// TwinCAT 3 PLC project database_connection
// Title: cyclic_database_recorder
// Company: Beckhoff K.K. - Japan
// Author: Takashi Ichihashi
// ProjectVersion: 1.0.1.1
// Description: The database recording library for InfluxDB. Requirements: Tc2_Utilities / T_Arg function
// ProgramVersion: 3.1.4023.0
// libraries:
//   Tc2_EtherCAT, * (Beckhoff Automation GmbH)
//   Tc2_Standard, * (Beckhoff Automation GmbH)
//   Tc2_System, * (Beckhoff Automation GmbH)
//   Tc2_Utilities, * (Beckhoff Automation GmbH)
//   Tc3_Database, * (Beckhoff Automation GmbH)
//   Tc3_IPCDiag, * (Beckhoff Automation GmbH)
//   Tc3_Module, * (Beckhoff Automation GmbH)
// project tree:
//   / DBWrite.TcTTO, PlcTask.TcTTO
//   DUTs/ ChunkCommand.TcDUT, DatabaseThroughput.TcDUT, DatabaseThroughput_SQL.TcDUT, DataTag.TcDUT, E_DbLogState.TcDUT, PerformanceData.TcDUT, ProcessModeData.TcDUT, RecordDataStructureInfo.TcDUT, SQLPerformanceData.TcDUT
//   GVLs/ GVL.TcGVL, DBLibParam.TcGVL
//   POUs/ DatabaseRecord.TcPOU, SampleProgram.TcPOU
//   POUs/library/ BufferedRecord.TcPOU, dequeue.TcPOU
//   POUs/library/InfluxDB/ InfluxdbMeasurement.TcPOU, RecordInfluxDB.TcPOU
//   POUs/library/interface/ IRecordDataQueue.TcIO, IRecordDB.TcIO
//   POUs/library/SQL/ FB_DatetimeUtilities.TcPOU, sql_parameters.TcPOU, RecordSQL.TcPOU
//   Project Information/ F_GetCompany.TcPOU, F_GetTitle.TcPOU, F_GetVersion.TcPOU
//   Version/ Global_Version.TcGVL
// real-time tasks:
//   TASK PlcTask: cycle T#1ms, priority 20, ADS port 350
//   TASK DBWrite: cycle T#10ms, priority 1, ADS port 351

CONFIGURATION database_connection
    RESOURCE PLC ON TwinCAT3
        TASK DBWrite(INTERVAL := T#10ms, PRIORITY := 1);
        TASK PlcTask(INTERVAL := T#1ms, PRIORITY := 20);
        PROGRAM DatabaseRecord WITH DBWrite : DatabaseRecord;
        PROGRAM SampleProgram WITH PlcTask : SampleProgram;
    END_RESOURCE
END_CONFIGURATION

// ---- DUTs/ChunkCommand.TcDUT
TYPE ChunkCommand :
STRUCT
	accumulated_amount: REFERENCE TO UDINT;
	chunk_size :UDINT;
	cycle_time_100ns : UDINT;
	start_time : ULINT;
	start_pointer : PVOID;
	structure_size : UDINT;
	structure_name : T_MaxString;
	sql_parameters: REFERENCE TO sql_parameters;
END_STRUCT
END_TYPE

// ---- DUTs/DatabaseThroughput.TcDUT
TYPE DatabaseThroughput:
STRUCT
	{attribute 'TagName' := 'machine_id'}
    machine_id : STRING(255); // 設備名
    {attribute 'TagName' := 'data_type_id'}
    job_id : STRING(255); // 発生イベント種別
	{attribute 'FieldName' := 'DB_queue_count'}
    db_insert_queue_count: UDINT;
	{attribute 'FieldName' := 'DB_buffer_current_index'}
    current_index: UDINT;
	{attribute 'FieldName' := 'DB_buffer_next_index'}
    next_index: UDINT;
	{attribute 'FieldName' := 'DB_buffer_usage'}
	buffer_usage: REAL;
END_STRUCT
END_TYPE

// ---- DUTs/DatabaseThroughput_SQL.TcDUT
TYPE DatabaseThroughput_SQL:
STRUCT
    datetime : ULINT; // UNIX epoch
    db_insert_queue_count: UDINT; // キューインされた一括インサート予定のコマンド数
    current_index: UDINT; // 現在のデータバッファの開始インデックス
    next_index: UDINT; // 次回インサートコマンドが発行される予定のバッファの終端インデックス
	buffer_usage: REAL; // バッファの使用率（全バッファサイズうのうちインサートコマンドが発行待ちのデータ数）
END_STRUCT
END_TYPE

// ---- DUTs/DataTag.TcDUT
(*
:作成日: 2023/3/1
:開発者: 市橋 卓

TF6420 database serverを用いた、influxDBのMeasurementにデータを書き込む際のタグ部分の構造体です。タグを定義する構造体は :ref:`figure_data_structure` に示す通り、フィールドを定義する構造体により継承されます。 

.. figure:: ../../LibraryBundle/data_struct.svg
    :width: 250px
    :align: center
    :name: figure_data_structure

    influxDBのデータタグの格納用構造体定義
	
*)
TYPE DataTag:
STRUCT
	{attribute 'TagName' := 'machine_id'}
    machine_id : STRING(255); // 設備名
    {attribute 'TagName' := 'data_type_id'}
    job_id : STRING(255); // 発生イベント種別
END_STRUCT
END_TYPE

// ---- DUTs/E_DbLogState.TcDUT
{attribute 'qualified_only'}
{attribute 'strict'}
TYPE E_DbLogState :
(
	idle := 0, 	// Buffer queing
    init,		// Not used
    writing,	// Writing to database
    error		// Get error response from database
);
END_TYPE

// ---- DUTs/PerformanceData.TcDUT
TYPE PerformanceData EXTENDS DataTag:
STRUCT
	{attribute 'FieldName' := 'plc_task_time'}
    task_time: UDINT;
	{attribute 'FieldName' := 'cpu_usage'}
    cpu_usage: UDINT;
	{attribute 'FieldName' := 'latency'}
    latency: UDINT;
	{attribute 'FieldName' := 'max_latency'}
    max_latency: UDINT;
	{attribute 'FieldName' := 'exceed_counter'}
    exceed_counter: UDINT;
	{attribute 'FieldName' := 'ec_lost_frames'}
    ec_lost_frames: UDINT;
	{attribute 'FieldName' := 'ec_frame_rate'}
    ec_frame_rate: LREAL;
	{attribute 'FieldName' := 'ec_lost_q_frame'}
    ec_lost_q_frames: UDINT;
	{attribute 'FieldName' := 'ec_q_frame_rate'}
    ec_q_frame_rate: LREAL;
END_STRUCT
END_TYPE

// ---- DUTs/ProcessModeData.TcDUT
TYPE ProcessModeData EXTENDS DataTag:
STRUCT
	{attribute 'FieldName' := 'executing'}
    executing: BOOL;
	{attribute 'FieldName' := 'message'}
	message: STRING := 'ABC000';
END_STRUCT
END_TYPE

// ---- DUTs/RecordDataStructureInfo.TcDUT
TYPE RecordDataStructureInfo :
STRUCT
	structure_pointer : PVOID;
	structure_size : UDINT;
	buffer_size :UDINT := DBLibParam.DATA_BUFFER_SIZE;
	structure_name : T_MaxString;
END_STRUCT
END_TYPE

// ---- DUTs/SQLPerformanceData.TcDUT
TYPE SQLPerformanceData :
STRUCT
	time_stamp: DT;
	task_time: DINT;
	cpu_usage: DINT;
	latency: DINT;
	max_latency: DINT;
	exceed_counter: DINT;
    db_insert_queue_count: DINT;
    current_index: DINT;
    next_index: DINT;
	buffer_usage: REAL;
END_STRUCT
END_TYPE

// ---- GVLs/GVL.TcGVL
{attribute 'qualified_only'}
VAR_GLOBAL
	// Database record driver
	fbInfluxDBRecorder	:RecordInfluxDB(DBID := 1);
	fbSQLRecorder 		:RecordSQL(DBID := 2);
END_VAR

// ---- GVLs/DBLibParam.TcGVL
{attribute 'qualified_only'}
VAR_GLOBAL CONSTANT
	COMMAND_QUEUE_BUFFER_SIZE :UDINT := 64; // Queue size for database insert command.
	DATA_BUFFER_SIZE	:UDINT := 500; // Data buffer size
	MAX_COLUMN_NUM		: UDINT := 50;
END_VAR

// ---- Version/Global_Version.TcGVL
{attribute 'TcGenerated'}
{attribute 'no-analysis'}
{attribute 'linkalways'}
// This function has been automatically generated from the project information.
VAR_GLOBAL CONSTANT
	{attribute 'const_non_replaced'}
	stLibVersion_cyclic_database_recorder : ST_LibVersion := (iMajor := 1, iMinor := 0, iBuild := 1, iRevision := 1, nFlags := 0, sVersion := '1.0.1.1');
END_VAR

// ---- POUs/library/interface/IRecordDataQueue.TcIO
INTERFACE IRecordDataQueue

(* Usage of data buffer (0 - 1.0) [1/100%] *)
PROPERTY PUBLIC buffer_usage : REAL
GET
END_GET
END_PROPERTY

(* Current index of data buffer array *)
PROPERTY index : UDINT
GET
END_GET
END_PROPERTY

PROPERTY PUBLIC max_chunk_size : UDINT
GET
END_GET
SET
END_SET
END_PROPERTY

PROPERTY PUBLIC min_chunk_size : UDINT
GET
END_GET
SET
END_SET
END_PROPERTY

(* The target buffer index at which assume the data in buffer reaches specified size and bulk insert command be sent to database engine.  *)
PROPERTY next_index : UDINT
GET
END_GET
END_PROPERTY

PROPERTY recorder : IRecordDB
GET
END_GET
SET
END_SET
END_PROPERTY

PROPERTY SQL_parameters : REFERENCE TO sql_parameters
GET
END_GET
END_PROPERTY

METHOD write : BOOL
VAR_INPUT
	input_data	:PVOID;
END_VAR
END_METHOD

END_INTERFACE

// ---- POUs/library/interface/IRecordDB.TcIO
INTERFACE IRecordDB

PROPERTY queue : REFERENCE TO dequeue
GET
END_GET
SET
END_SET
END_PROPERTY

END_INTERFACE

// ---- POUs/DatabaseRecord.TcPOU
PROGRAM DatabaseRecord
VAR
	test : FB_MemRingBuffer;
END_VAR

// Database Writing actions
GVL.fbInfluxDBRecorder();
GVL.fbSQLRecorder();

END_PROGRAM

// ---- POUs/SampleProgram.TcPOU
(*

Record performance data to influxDB and ANY SQL database
--------------------------------------------------------


* Objects

   Item List:
   
       This is body of item lists
	   
   Second Item:

      This is body of second items.
	  
	  
History
=====================

.. csv-table::
	:header: Rev., Date,Description
	
	0, 2023-01-10,Initial edition
	1, 2023-02-27,Add reStructuredText
	2, 2024-06-01,Add SQL database support
	  
*)

PROGRAM SampleProgram

VAR CONSTANT
	RECORD_DATA_MAX_INDEX: UDINT := 49999;
END_VAR

VAR
	
	// Initial
	initialized : BOOL;
	
	// Datetime utilities
	fbDtUtil : FB_DatetimeUtilities;

	// PLC System parameters
    fbGetCurTaskIdx  : GETCURTASKINDEX;
	test_timer :TON; // Inclese workload rate
	bExecuting :BOOL;
	j:UDINT := 0;
	target: UDINT := 5000;
	test_var:ULINT;
	
	process_timer :TON; // Process time

	// for InfluxDB

	// Record data buffer
	DatabaseThroughputRecordData 		:DatabaseThroughput;	// for insert dataset
	DatabaseThroughputRecordBuffer 		:ARRAY [0..DBLibParam.DATA_BUFFER_SIZE] OF DatabaseThroughput;

	fbThroughputRecorder_influxDB		:BufferedRecord(
												GVL.fbInfluxDBRecorder, 
												ADR(DatabaseThroughputRecordBuffer)
										);		// record controller

	// For SQL DB

	// Record data buffer
	DatabaseThroughputRecordData_SQL 		:DatabaseThroughput_SQL;	// for insert dataset
	DatabaseThroughputRecordBuffer_SQL 		:ARRAY [0..DBLibParam.DATA_BUFFER_SIZE] OF DatabaseThroughput_SQL;

	fbThroughputRecorder_SQLDB			:BufferedRecord(
												GVL.fbSQLRecorder, 
												ADR(DatabaseThroughputRecordBuffer_SQL)
										);		// record controller

END_VAR

(* Initialize*)
IF NOT initialized THEN
	// Influx DB
	fbThroughputRecorder_influxDB.set_buffer_info(
		struct_size := SIZEOF(DatabaseThroughputRecordBuffer[0]),
		buffer_size := SIZEOF(DatabaseThroughputRecordBuffer),
		structure_name := 'DatabaseThroughput'); // Measurement name
	fbThroughputRecorder_influxDB.SQL_parameters.table_name := 'DatabaseThroughput'; // Structure type name
	// SQL DB
	fbThroughputRecorder_SQLDB.set_buffer_info(
		struct_size := SIZEOF(DatabaseThroughputRecordBuffer_SQL[0]),
		buffer_size := SIZEOF(DatabaseThroughputRecordBuffer_SQL),
		structure_name := ''); // Measurement name
	fbThroughputRecorder_SQLDB.SQL_parameters.table_name := 'database_throughput';
	fbThroughputRecorder_SQLDB.SQL_parameters.add_column('datetime', E_ExpParameterType.Int64, SIZEOF(DatabaseThroughputRecordData_SQL.datetime));
	fbThroughputRecorder_SQLDB.SQL_parameters.add_column('db_insert_queue_count', E_ExpParameterType.Int32, SIZEOF(DatabaseThroughputRecordData_SQL.db_insert_queue_count));
	fbThroughputRecorder_SQLDB.SQL_parameters.add_column('current_index', E_ExpParameterType.Int32, SIZEOF(DatabaseThroughputRecordData_SQL.current_index));
	fbThroughputRecorder_SQLDB.SQL_parameters.add_column('next_index', E_ExpParameterType.Int32, SIZEOF(DatabaseThroughputRecordData_SQL.next_index));
	fbThroughputRecorder_SQLDB.SQL_parameters.add_column('buffer_usage', E_ExpParameterType.Float32, SIZEOF(DatabaseThroughputRecordData_SQL.buffer_usage));
	initialized := TRUE;
END_IF


fbDtUtil();


(*
	Database Throughput data insert buffer
*)


(* Data set here *)
// cyclic record > influxdb

// Tag Data
DatabaseThroughputRecordData.machine_id := 'machine-1';
DatabaseThroughputRecordData.job_id := 'db_throughput';
// Field data
DatabaseThroughputRecordData.db_insert_queue_count := GVL.fbInfluxDBRecorder.queue.queue_usage;
DatabaseThroughputRecordData.current_index := fbThroughputRecorder_influxDB.index;
DatabaseThroughputRecordData.next_index := fbThroughputRecorder_influxDB.next_index;
DatabaseThroughputRecordData.buffer_usage := fbThroughputRecorder_influxDB.buffer_usage;

(* Queue set *)
fbThroughputRecorder_influxDB.write(ADR(DatabaseThroughputRecordData));

// cyclic record > SQLdb
DatabaseThroughputRecordData_SQL.datetime := fbDtUtil.Filetime_To_UnixT(F_GetSystemTime());
DatabaseThroughputRecordData_SQL.db_insert_queue_count := GVL.fbSQLRecorder.queue.queue_usage;
DatabaseThroughputRecordData_SQL.current_index := fbThroughputRecorder_SQLDB.index;
DatabaseThroughputRecordData_SQL.next_index := fbThroughputRecorder_SQLDB.next_index;
DatabaseThroughputRecordData_SQL.buffer_usage := fbThroughputRecorder_SQLDB.buffer_usage;

fbThroughputRecorder_SQLDB.write(ADR(DatabaseThroughputRecordData_SQL));

END_PROGRAM

// ---- POUs/library/SQL/FB_DatetimeUtilities.TcPOU
FUNCTION_BLOCK FB_DatetimeUtilities
VAR_INPUT
END_VAR
VAR_OUTPUT
END_VAR
VAR
	sPrintf : FB_FormatString;
	fbTZInfo : FB_GetTimeZoneInformation;
	check_interval : TON;
	check_event :BOOL := TRUE;
END_VAR

check_interval(IN := NOT check_interval.Q, PT := T#15M);

IF check_interval.Q THEN
	check_event := TRUE;
END_IF

fbTZInfo(bExecute := check_event);

IF check_event AND NOT fbTZInfo.bBusy THEN
	check_event := FALSE;
END_IF

METHOD Filetime_To_Timestamp : T_MaxString
VAR_INPUT
	datetime : T_filetime64;
END_VAR
VAR
	dc_time : DCTIMESTRUCT;
	bias : DINT;
END_VAR


dc_time := DCTIME64_TO_DCTIMESTRUCT(FILETIME64_TO_DCTIME64(datetime));
bias := fbTZInfo.tzInfo.bias / 60;

sPrintf(sFormat := '%.4d-%.2d-%.2d %.2d:%.2d:%.2d.%.3d%.3d%.2d',
        arg1 := F_WORD(dc_time.wYear),
        arg2 := F_WORD(dc_time.wMonth),
        arg3 := F_WORD(dc_time.wDay),
        arg4 := F_WORD(dc_time.wHour),
        arg5 := F_WORD(dc_time.wMinute),
        arg6 := F_WORD(dc_time.wSecond),
        arg7 := F_WORD(dc_time.wMilliseconds),
		arg8 := F_WORD(dc_time.wMicroseconds),
		arg9 := F_DINT(bias)
);

Filetime_To_Timestamp := sPrintf.sOut;
END_METHOD

METHOD Filetime_To_UnixT : ULINT
VAR_INPUT
	datetime : T_filetime64;
END_VAR
Filetime_To_UnixT := (datetime - 116444736000000000) / 10;
END_METHOD

END_FUNCTION_BLOCK

// ---- POUs/library/BufferedRecord.TcPOU
(*
Bufferd mode that is accumulated and bulk insert. Accumulated data size is calculated automatically among mininum/maximum_chunk_size parameter.
*)

FUNCTION_BLOCK BufferedRecord IMPLEMENTS IRecordDataQueue
VAR
	_current_index	: UDINT; // current index value
	_next_index 		: UDINT;
	_min_chunk_size				: UDINT := DBLibParam.DATA_BUFFER_SIZE / 20;		// Minimum chunk size
	_max_chunk_size				: UDINT	:= DBLibParam.DATA_BUFFER_SIZE;				// Maximum chunk size
	_buffer_byte_size			: UDINT;
	_buffer_array_size			: UDINT;			// upper bound of data buffer array.
	_buffer_usage				: REAL;				// data usage percentage of data buffer.
	_buffer_pointer 			: PVOID := 0;
	_sql_parameters				: sql_parameters;
	_structure_pointer : PVOID;
	_structure_size : UDINT;
	_structure_name : T_MaxString;
	_recorder 					: IRecordDB;
END_VAR

{warning 'add property implementation'}
(* Usage of data buffer (0 - 1.0) [1/100%] *)
PROPERTY buffer_usage : REAL
GET
buffer_usage := _buffer_usage;
END_GET
END_PROPERTY

METHOD FB_init : BOOL
VAR_INPUT
	bInitRetains : BOOL; // if TRUE, the retain variables are initialized (warm start / cold start)
	bInCopyCode : BOOL;  // if TRUE, the instance afterwards gets moved into the copy code (online change)
	recorder	:IRecordDB; // IRecordDB is a interface class of database connection endpoint object.
	buffer_pointer	: PVOID;
END_VAR
_recorder := recorder;
_buffer_pointer := buffer_pointer;
END_METHOD

(* Current index of data buffer array *)
PROPERTY index : UDINT
GET
index := _current_index;
END_GET
END_PROPERTY

PROPERTY PUBLIC max_chunk_size : UDINT
GET
max_chunk_size := _max_chunk_size;
END_GET
SET
_max_chunk_size := max_chunk_size;
END_SET
END_PROPERTY

PROPERTY PUBLIC min_chunk_size : UDINT
GET
min_chunk_size := _min_chunk_size;
END_GET
SET
_min_chunk_size := min_chunk_size;
END_SET
END_PROPERTY

(* The target buffer index at which assume the data in buffer reaches specified size and bulk insert command be sent to database engine.  *)
PROPERTY next_index : UDINT
GET
next_index := _next_index;
END_GET
END_PROPERTY

{warning 'add property implementation'}
PROPERTY recorder : IRecordDB
GET
recorder := _recorder;
END_GET
SET
_recorder := recorder;
END_SET
END_PROPERTY

METHOD set_buffer_info : BOOL
VAR_INPUT
	struct_size: UDINT;
	buffer_size : UDINT;
	structure_name: STRING;
END_VAR
_buffer_byte_size := buffer_size;
_structure_size := struct_size;
_buffer_array_size := buffer_size / struct_size;
_structure_name := structure_name;
END_METHOD

{warning 'add property implementation'}
PROPERTY SQL_parameters : REFERENCE TO sql_parameters
GET
SQL_parameters REF= _sql_parameters;
END_GET
END_PROPERTY

(*The method to write to database through data buffer with queue.*)
{warning 'add method implementation '}
METHOD write : BOOL // Return true if data is put on buffer queue successfully.
VAR_INPUT
	input_data	: PVOID;	// Set the measured data. It should be same data type as item of data buffer that is set at "buffer_pointer" on "FB_init" constructor.
END_VAR
VAR
	gCurrentData	:T_Arg;
	pCurrentBufferPointer : PVOID;
	work_data_body  :ChunkCommand;
	nTaskIdx: DINT;
	queue_input_flag: BOOL;
END_VAR
VAR_INST
// Start point time
	start_time		: ULINT;
	start_data 		: T_Arg;

	nCycleTime		: UDINT;					// PLC task cycle time setting(in 100ns)
	data_size		: UDINT := 1;				// record data size
	accumulated_amount		: UDINT := 0;		// buffer usage
	last_data_count	: UDINT := 0;
	
	start_index		: UDINT;
	_avalable_buffer_size	:DINT;
	diff_target		: REAL;
	pid_ope			: REAL;	
	chunk_size 		: UDINT;
END_VAR
IF _recorder = 0 THEN
	write := FALSE;
	RETURN;
END_IF

pCurrentBufferPointer := _buffer_pointer + _structure_size * _current_index;
MEMCPY(pCurrentBufferPointer, input_data, _structure_size);
gCurrentData := F_BIGTYPE(pData := pCurrentBufferPointer, cbLen := _structure_size);

IF _current_index = start_index THEN
	start_time := F_GetSystemTime();
	start_data := gCurrentData;
END_IF

queue_input_flag := FALSE;

IF _next_index <= _current_index OR _current_index >= (_buffer_array_size - 1 ) THEN
	//max_chunk_size := nDataBufferMaxIndex + 1;
	// put_data
	IF NOT _recorder.queue.full THEN
		data_size := _current_index - start_index + 1;
		_avalable_buffer_size := UDINT_TO_DINT(_buffer_array_size) - UDINT_TO_DINT(accumulated_amount);
		IF _avalable_buffer_size < UDINT_TO_DINT(data_size) AND _avalable_buffer_size > 0 THEN
			data_size := DINT_TO_UDINT(_avalable_buffer_size);
		ELSIF _avalable_buffer_size <= 0 THEN
			data_size := 0;
		END_IF

		IF data_size > 1 THEN			
			// calculate each cycle time by num of data among start time and current time.
			nCycleTime := ULINT_TO_UDINT(F_GetSystemTime() - start_time) / (data_size - 1);
		ELSE
			nTaskIdx := GETCURTASKINDEXEX();
			IF nTaskIdx > 0 THEN
				nCycleTime := TwinCAT_SystemInfoVarList._TaskInfo[nTaskIdx].CycleTime;
			END_IF
		END_IF
		
		work_data_body.start_pointer := start_data.pData;
		work_data_body.start_time := start_time;
		work_data_body.cycle_time_100ns := nCycleTime;
		work_data_body.chunk_size := data_size;
		work_data_body.accumulated_amount REF= accumulated_amount;
		work_data_body.structure_size := _structure_size;
		work_data_body.structure_name := _structure_name;
		work_data_body.sql_parameters REF= _sql_parameters;
		// queue in
		_recorder.queue.put(work_data_body);
		start_index := _current_index + 1;
		queue_input_flag := TRUE;
	END_IF
END_IF


IF last_data_count <> accumulated_amount OR queue_input_flag THEN
	(*Re-calculate chunk size when amount of buffered data is changed including dequeued by recorder.*)
	// calculate next index
	_buffer_usage := UDINT_TO_REAL(accumulated_amount) / UDINT_TO_REAL(_buffer_array_size);
	diff_target := UDINT_TO_REAL(_max_chunk_size) * _buffer_usage;
	pid_ope := UDINT_TO_REAL(_min_chunk_size) + diff_target;
	chunk_size := REAL_TO_UDINT(pid_ope);
	IF chunk_size < _min_chunk_size OR pid_ope < 0 THEN
		chunk_size := _min_chunk_size;
	ELSIF chunk_size > _max_chunk_size THEN
		chunk_size := _max_chunk_size;
	END_IF
	//chunk_size := minimum_chunk_size;
	_next_index := _current_index + chunk_size;
END_IF

last_data_count := accumulated_amount;

IF _current_index < _buffer_array_size - 1 THEN
	_current_index := _current_index + 1;
ELSE
	_current_index := 0;
	start_index := 0;
	_next_index := chunk_size - 1;
END_IF

write := TRUE;
END_METHOD

END_FUNCTION_BLOCK

// ---- POUs/library/SQL/sql_parameters.TcPOU
FUNCTION_BLOCK sql_parameters
VAR_INPUT
END_VAR
VAR_OUTPUT
END_VAR
VAR
	_parameter : ARRAY [0..DbLibParam.MAX_COLUMN_NUM - 1] OF ST_ExpParameter;
	_table_name : STRING;
	current_column_index : UDINT := 0;
END_VAR

{warning 'add method implementation '}
METHOD add_column : BOOL
VAR_INPUT
	sParaName : T_MaxString;
	eParaType : E_ExpParameterType;
	nParaSize : UDINT;
END_VAR
IF DbLibParam.MAX_COLUMN_NUM < current_column_index THEN
	add_column := FALSE;
	RETURN;
END_IF 
_parameter[current_column_index].sParaName := sParaName;
_parameter[current_column_index].eParaType := eParaType;
_parameter[current_column_index].nParaSize := nParaSize;
current_column_index := current_column_index + 1;
add_column := TRUE;
END_METHOD

{warning 'add property implementation'}
PROPERTY cbParameters : UDINT
GET
IF current_column_index = 0 THEN
	cbParameters := 0;
ELSE
	cbParameters := SIZEOF(_parameter[0]) * current_column_index;
END_IF
END_GET
END_PROPERTY

{warning 'add property implementation'}
PROPERTY column_num : UDINT
GET
column_num := current_column_index;
END_GET
END_PROPERTY

{warning 'add property implementation'}
PROPERTY insert_query_string : Tc2_System.T_MaxString
GET
VAR
	i : UDINT;
END_VAR
insert_query_string := 'INSERT INTO ';
insert_query_string := CONCAT(insert_query_string, _table_name);
insert_query_string := CONCAT(insert_query_string, ' (');
FOR i := 0 TO current_column_index - 1 DO
	IF i > 0 THEN
		insert_query_string := CONCAT(insert_query_string,', ');	
	END_IF
	//insert_query_string := CONCAT(insert_query_string,'[');
	insert_query_string := CONCAT(insert_query_string,_parameter[i].sParaName);
	//insert_query_string := CONCAT(insert_query_string,']');
END_FOR
insert_query_string := CONCAT(insert_query_string, ')');
insert_query_string := CONCAT(insert_query_string, ' VALUES (');
FOR i := 0 TO current_column_index - 1 DO
	IF i > 0 THEN
		insert_query_string := CONCAT(insert_query_string,', ');
	END_IF
	insert_query_string := CONCAT(insert_query_string,'{');
	insert_query_string := CONCAT(insert_query_string,_parameter[i].sParaName);
	insert_query_string := CONCAT(insert_query_string,'}');
END_FOR
insert_query_string := CONCAT(insert_query_string, ');');
END_GET
END_PROPERTY

{warning 'add property implementation'}
PROPERTY pParameters : PVOID
GET
pParameters := ADR(_parameter[0]);
END_GET
END_PROPERTY

{warning 'add property implementation'}
PROPERTY table_name : STRING
GET
table_name := _table_name;
END_GET
SET
_table_name := table_name;
END_SET
END_PROPERTY

END_FUNCTION_BLOCK

// ---- POUs/library/InfluxDB/RecordInfluxDB.TcPOU
(*
Insert dedicated driver for InfluxDB.

:Author: 

	Takashi Ichihashi Beckhoff Automation K.K.
	
:Date:

	2023-03-09
	
This function block is based on sample code published on infosys sites. 
Link:  `https://infosys.beckhoff.com/content/1033/tf6420_tc3_database_server/8117583755.html?id=5199556541044360835 <https://infosys.beckhoff.com/content/1033/tf6420_tc3_database_server/8117583755.html?id=5199556541044360835>`

	
*)

FUNCTION_BLOCK RecordInfluxDB IMPLEMENTS IRecordDB

VAR_OUTPUT
	bBusy			: BOOL;	// In writing database
	bError			: BOOL; // Somthing wrong situation happend
	TcResult		: Tc3_Database.I_TcMessage; // Response message
    sErrorMessage	: STRING(255);	// Error message
END_VAR
VAR
	QueryOption_TSDB_Insert 			: T_QueryOptionTimeSeriesDB_Insert; // defines detailed Queryparameter
    fbNoSQLQueryBuilder_TimeSeriesDB 	: FB_NoSQLQueryBuilder_TimeSeriesDB; // defines database type specific api
    fbNoSqlQueryEvt 					: FB_NoSQLQueryEvt(sNetID := '', tTimeout := T#15S); // functionblock to execute queries
	
	// Variables for queue feature
	get_data 			: ChunkCommand;
	State				: E_DbLogState;
	_dbid				: UDINT;
	_queue : dequeue;	
END_VAR

CASE State OF

	E_DbLogState.idle:
		
		IF NOT fbNoSqlQueryEvt.bBusy THEN
			State := E_DbLogState.init;
		END_IF

	E_DbLogState.init:
	
		IF NOT fbNoSqlQueryEvt.bBusy AND _queue.queue_usage > 0 THEN
			// getting data
			get_data := _queue.get();
			// Data set
			IF get_data.chunk_size > 0 THEN
				fbNoSQLQueryBuilder_TimeSeriesDB.pQueryOptions := ADR(QueryOption_TSDB_Insert);
				fbNoSQLQueryBuilder_TimeSeriesDB.cbQueryOptions := SIZEOF(QueryOption_TSDB_Insert);    
				QueryOption_TSDB_Insert.sTableName := get_data.sql_parameters.table_name;
				QueryOption_TSDB_Insert.sDataType := get_data.structure_name;
				QueryOption_TSDB_Insert.pSymbol := get_data.start_pointer;
				QueryOption_TSDB_Insert.cbSymbol := get_data.structure_size * get_data.chunk_size;
				QueryOption_TSDB_Insert.nDataCount := get_data.chunk_size;
				QueryOption_TSDB_Insert.nStartTimestamp := get_data.start_time;
				QueryOption_TSDB_Insert.nCycleTime := get_data.cycle_time_100ns; // (in 100 ns)
				State := E_DbLogState.writing;
			END_IF
		
		END_IF

	E_DbLogState.writing:
	
		IF fbNoSqlQueryEvt.Execute(_dbid, fbNoSQLQueryBuilder_TimeSeriesDB) THEN
			IF fbNoSqlQueryEvt.bError THEN
				TcResult := fbNoSqlQueryEvt.ipTcResult;                
				State := E_DbLogState.error;
			ELSE		
				State := E_DbLogState.idle;
				bError := FALSE;
			END_IF
		END_IF

	E_DbLogState.error:
	
		IF TcResult.RequestEventText(1033, sErrorMessage, SIZEOF(sErrorMessage)) THEN
            TcResult.Send(F_GetSystemTime());
            State := E_DbLogState.idle;
            bError := TRUE;
        END_IF
END_CASE

METHOD FB_init : BOOL
VAR_INPUT
	bInitRetains : BOOL; // if TRUE, the retain variables are initialized (warm start / cold start)
	bInCopyCode : BOOL;  // if TRUE, the instance afterwards gets moved into the copy code (online change)
	DBID		: UDINT; //Database ID for TF6420 configurator
END_VAR
_dbid := DBID;
END_METHOD

(*Property of database command queue*)
{warning 'add property implementation'}
PROPERTY queue : REFERENCE TO dequeue
GET
queue REF= _queue;
END_GET
SET
_queue := queue;
END_SET
END_PROPERTY

END_FUNCTION_BLOCK

// ---- POUs/library/dequeue.TcPOU
(*
:Author: Takashi Ichihashi
:Date: 2023-03-07

Decreration
=========================

.. code-block:: 

	// Variables for queue feature
	fb_deq : dequeue;
	get_data : T_Arg;
	// databuffer for 1 second with 10 ms time delta
    queue_buffer: ARRAY[0..99] OF T_Arg;
	

Useage
=================

This is example code that the sInputData is queued in and queued out for sOutputData.

.. code-block:: 

	// put_data
	IF NOT fb_deq.full THEN

		sInputData := ANY_DATA;
		// put pointer
		fb_deq.put(F_BIGTYPE(ADR(sInputData),SIZEOF(sInputData)));

	END_IF
	
	// getting data
	get_data := fb_deq.get();
	MEMCPY(ADR(sOutputData), get_data.pData, get_data.cbLen);
	
	
*)

FUNCTION_BLOCK dequeue
VAR
	_queue_usage:	UDINT;
	_queue_size:	UDINT := DbLibParam.COMMAND_QUEUE_BUFFER_SIZE;
	nWriteIndex: 	UDINT;
	nReadIndex: 	UDINT;
	queue_buffer:	ARRAY [0..DbLibParam.COMMAND_QUEUE_BUFFER_SIZE - 1] OF ChunkCommand;
END_VAR

PROPERTY full : BOOL
GET
full :=  _queue_usage >= DBLibParam.COMMAND_QUEUE_BUFFER_SIZE - 1;
END_GET
END_PROPERTY

METHOD get : ChunkCommand
VAR_INPUT
END_VAR
//Set buffer index

IF _queue_usage > 0 THEN
	get := queue_buffer[nReadIndex];
	get.accumulated_amount := get.accumulated_amount - get.chunk_size;
	_queue_usage := _queue_usage - 1;
	nReadIndex := nReadIndex + 1;
	IF nReadIndex > DBLibParam.COMMAND_QUEUE_BUFFER_SIZE - 1 THEN
		nReadIndex := 0;
	END_IF
END_IF

RETURN;
END_METHOD

PROPERTY PUBLIC index : UDINT
GET
index := nWriteIndex;
END_GET
END_PROPERTY

PROPERTY PUBLIC max_index : UDINT
GET
max_index := DBLibParam.COMMAND_QUEUE_BUFFER_SIZE - 1;
END_GET
END_PROPERTY

METHOD PUBLIC put : UDINT
VAR_INPUT
	lData:	ChunkCommand;
END_VAR
//Set buffer index

IF _queue_usage >= DBLibParam.COMMAND_QUEUE_BUFFER_SIZE - 1 THEN
	put := 0;
ELSE
	queue_buffer[nWriteIndex] := lData;
	lData.accumulated_amount := lData.accumulated_amount + lData.chunk_size;
	_queue_usage := _queue_usage + 1;
	nWriteIndex := nWriteIndex + 1;
	IF nWriteIndex > DBLibParam.COMMAND_QUEUE_BUFFER_SIZE - 1 THEN
		nWriteIndex := 0;
	END_IF
	put := 1;
END_IF

RETURN;
END_METHOD

PROPERTY queue_size : UDINT
GET
queue_size := _queue_size;
END_GET
END_PROPERTY

PROPERTY queue_usage : UDINT
GET
queue_usage := _queue_usage;
END_GET
END_PROPERTY

END_FUNCTION_BLOCK

// ---- POUs/library/SQL/RecordSQL.TcPOU
(*

	
*)

FUNCTION_BLOCK RecordSQL IMPLEMENTS IRecordDB
VAR_OUTPUT
	bBusy			: BOOL;	// In writing database
	bError			: BOOL; // Somthing wrong situation happend
	TcResult		: Tc3_Database.I_TcMessage; // Response message
    sErrorMessage	: STRING(255);	// Error message
END_VAR
VAR
	
	//for generating timestamp
	fbGetSystemTime1: GetSystemTime;
	dwTimeLoDW: DWORD;
	dwTimeHiDW: DWORD;
	tFileTime: T_FILETIME;
	nTimestamp: LINT;
	
	//for insert samples
	fbPLCDBCmd: FB_PLCDBCmdEvt(sNetID := '', tTimeout := T#19S);

	// Variables for queue feature
	get_data 			: ChunkCommand;
	State				: E_DbLogState;
	_dbid				: UDINT;
	_queue 				: dequeue;	
	_query				: T_MaxString;
	pParam: PVOID;
	cbParam: UDINT;
END_VAR


CASE State OF

	E_DbLogState.idle:
		
		IF NOT fbPLCDBCmd.bBusy THEN
			State := E_DbLogState.init;
		END_IF

	E_DbLogState.init:
	
		IF NOT fbPLCDBCmd.bBusy AND _queue.queue_usage > 0 THEN
			// getting data
			get_data := _queue.get();
			_query := get_data.sql_parameters.insert_query_string;
			State := E_DbLogState.writing;
		END_IF

	E_DbLogState.writing:
		pParam := get_data.sql_parameters.pParameters;
		cbParam := get_data.sql_parameters.cbParameters;
		
		//Write buffer element to database
		IF fbPLCDBCmd.Execute(_dbid, 
							ADR(_query), 
							SIZEOF(_query), 
							get_data.start_pointer, 
							get_data.structure_size * get_data.chunk_size, 
							pParam, 
							cbParam) THEN
			IF fbPLCDBCmd.bError THEN
				State := E_DbLogState.error;
			ELSE
				State := E_DbLogState.init;
			END_IF				
		END_IF
		

	E_DbLogState.error:
		//IF TcResult.RequestEventText(1033, sErrorMessage, SIZEOF(sErrorMessage)) THEN
            //TcResult.Send(F_GetSystemTime());
            State := E_DbLogState.idle;
            bError := TRUE;
        //END_IF

END_CASE

{warning 'add method implementation '}
METHOD FB_init : BOOL
VAR_INPUT
	(* if TRUE, the retain variables are initialized (warm start / cold start)*)
	bInitRetains	: BOOL;
	(* if TRUE, the instance afterwards gets moved into the copy code (online change)*)
	bInCopyCode	: BOOL;
	(*Database ID for TF6420 configurator*)
	DBID	: UDINT;
END_VAR
_dbid := DBID;
END_METHOD

{warning 'add property implementation'}
PROPERTY queue : REFERENCE TO dequeue
GET
queue REF= _queue;
END_GET
SET
_queue := queue;
END_SET
END_PROPERTY

END_FUNCTION_BLOCK

// ---- POUs/library/InfluxDB/InfluxdbMeasurement.TcPOU
FUNCTION_BLOCK InfluxdbMeasurement IMPLEMENTS InterfaceSQLParameters
VAR_INPUT
END_VAR
VAR_OUTPUT
END_VAR
VAR
	_measurement_name :T_MaxString;
END_VAR

{warning 'add method implementation '}
METHOD add_column : BOOL
VAR_INPUT
	paramater	: Tc3_Database.ST_ExpParameter;
END_VAR
END_METHOD

{warning 'add property implementation'}
PROPERTY cbParameters : UDINT
GET
END_GET
END_PROPERTY

{warning 'add property implementation'}
PROPERTY column_num : UDINT
GET
END_GET
END_PROPERTY

{warning 'add property implementation'}
PROPERTY insert_query_string : Tc2_System.T_MaxString
GET
END_GET
END_PROPERTY

{warning 'add property implementation'}
PROPERTY pParameters : PVOID
GET
END_GET
END_PROPERTY

{warning 'add property implementation'}
PROPERTY table_name : Tc2_System.T_MaxString
GET
table_name := _measurement_name;
END_GET
SET
_measurement_name := table_name;
END_SET
END_PROPERTY

END_FUNCTION_BLOCK

// ---- Project Information/F_GetCompany.TcPOU
// This function has been automatically generated from the project information.
{attribute 'signature_flag' := '1073741824'}
{attribute 'TcGenerated'}
{attribute 'no-analysis'}
FUNCTION F_GetCompany : WSTRING
VAR_INPUT
	
END_VAR

F_GetCompany := "Beckhoff K.K. - Japan";

END_FUNCTION

// ---- Project Information/F_GetTitle.TcPOU
// This function has been automatically generated from the project information.
{attribute 'signature_flag' := '1073741824'}
{attribute 'TcGenerated'}
{attribute 'no-analysis'}
FUNCTION F_GetTitle : WSTRING
VAR_INPUT
	
END_VAR

F_GetTitle := "cyclic_database_recorder";

END_FUNCTION

// ---- Project Information/F_GetVersion.TcPOU
// This function has been automatically generated from the project information.
{attribute 'signature_flag' := '1073741824'}
{attribute 'TcGenerated'}
{attribute 'no-analysis'}
FUNCTION F_GetVersion : ST_LibVersion
VAR_INPUT
	
END_VAR

F_GetVersion.iMajor := 1;
F_GetVersion.iMinor := 0;
F_GetVersion.iBuild := 1;
F_GetVersion.iRevision := 1;
F_GetVersion.sVersion := '1.0.1.1';
F_GetVersion.nFlags := 0;

END_FUNCTION
